{region '#Template'}
	{attribute 'Category' := 'Universal'}
	{attribute 'Version' := '0.0.1.0'}
	{attribute 'Tags' := 'Universal, Analog, Aggregate'}
	{attribute 'Description' := 'Aktor analog	// Actuator analog'}
{endregion}	 
FUNCTION_BLOCK FB_BA_ActuatorAnalog EXTENDS FB_BA_AggregateA
VAR_OUTPUT
	fPresentValue			: REAL;
END_VAR
VAR_INPUT CONSTANT
	Mdlt					: FB_BA_AO_IO;
END_VAR
VAR
END_VAR

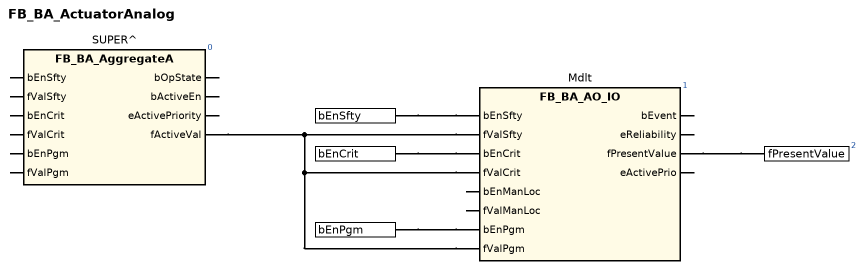
SUPER^(); // FB_BA_AggregateA
Mdlt(
    bEnSfty := bEnSfty,
    fValSfty := SUPER^.fActiveVal,
    bEnCrit := bEnCrit,
    fValCrit := SUPER^.fActiveVal,
    bEnPgm := bEnPgm,
    fValPgm := SUPER^.fActiveVal); // FB_BA_AO_IO
fPresentValue := Mdlt.fPresentValue;

METHOD FB_init : BOOL
VAR_INPUT
	bInitRetains : BOOL; // if TRUE, the retain variables are initialized (warm start / cold start)
	bInCopyCode : BOOL;  // if TRUE, the instance afterwards gets moved into the copy code (online change)
END_VAR
Mdlt.iParent					:= THIS^;
Mdlt.iLabel						:= LblUniFieldDevice.Aggregat_Mdlt;	
Mdlt.sObjectName				:= '{Idx=01}';
Mdlt.sDeviceType				:= '';
Mdlt.bEnOutOfService			:= FALSE;
Mdlt.eOverriddenPolarity		:= E_BA_Polarity.eNormal;
Mdlt.eUnit						:= E_BA_Unit.eOther_Percent;
Mdlt.fResolution 				:= 0.003051851;
Mdlt.fScaleOffset 				:= 0;
Mdlt.fCOVIncrement				:= BA2_Param.fDefCOVIncrement;
Mdlt.bEnManualRm				:= FALSE;	//	Priority  8	
Mdlt.fValManualRm				:= 0.0;		//	Priority  8
Mdlt.fDefaultValue				:= 0.0;	
Mdlt.nEventClassID				:= EventClasses.NotificationSimple;
Mdlt.stTimeDelay.nToNormal		:= BA2_Param.nDefTimeDelay_ToNormal;
Mdlt.stTimeDelay.nToAbnormal	:= BA2_Param.nDefTimeDelay_ToAbnormal;
Mdlt.stHighLimit.bEnable		:= FALSE;
Mdlt.stHighLimit.fValue			:= 0.0;		
Mdlt.stLowLimit.bEnable			:= FALSE;
Mdlt.stLowLimit.fValue			:= 0.0;
Mdlt.fLimitDeadband 			:= BA2_Param.fDefLimitDeadband;
Mdlt.bAcknowledgeRm				:= FALSE;	
Mdlt.aEventTransitionText[1]	:= Texts.txtDisturb;
Mdlt.aEventTransitionText[2]	:= Texts.txtNone;
Mdlt.aEventTransitionText[3]	:= Texts.txtNormal;
Mdlt.bEventDetectionEnable		:= FALSE;
Mdlt.eEnPlantLock				:= E_BA_LockPriority.eNoLock;
END_METHOD

END_FUNCTION_BLOCK

(* stored: Version 1.1.0.1, ProductVersion 3.1.4024.6
   POU FB_BA_ActuatorAnalog: Id {d5f27d11-ffa1-44e3-8cda-68bb166e0287}, SpecialFunc None
   Method FB_init: Id {86a40007-01ba-47e4-a71a-4e6cd603dd48} *)
